FUNCTION_BLOCK FB_GreenConveyor
VAR
	Motor					:FB_ConveyorMotor;
	LTU						:FB_LTU_Cylinder;	
    BlueStopper				:FB_Stopper;
    nStatus					:INT:=0;	
				
END_VAR

END_FUNCTION_BLOCK

(* stored: Version 1.1.0.1, ProductVersion 3.1.4024.12
   POU FB_GreenConveyor: Id {120bdc55-22e1-42a9-8b1f-b54ef0d19c05}, SpecialFunc None *)
